Staubli VAL3: start.pgx

program start()
  local num l_ncouleur_bout
begin

  //  sioCtrl(sData, "port", 8500)
  //  sioCtrl(sData, "clients", 1)
  //  //CCaractère de fin de line : Line Feed
  //  sioCtrl(sData, "endOfString", 13)

  //  logMsg("------------ Sio Initialise")

  //  logMsg("  dataAcquisition start")
  //  do

  //    nb=0
  //    i=0
  //    while(nb<32)
  //      nb=sioGet(sData, l_nByteIn[i])

  //      if(nb>0)
  //        i=i+nb
  //      else
  //        // Erreur de communication
  //        return
  //      endIf
  //      logMsg("Recuperation du buffer...")
  //    endWhile
  //    logMsg("Buffer récupéré.")



  l_ncouleur_bout=1

  call picketplace(l_ncouleur_bout)


  l_ncouleur_bout=0
  call picketplace(l_ncouleur_bout)
  waitEndMove()

end
